// TIA Portal V19 export
DATA_BLOCK "DB_CommSlave"   // DB40
{ S7_Optimized_Access := 'TRUE' }
// stored: AutoNumber false, MemoryReserve 100
   VAR
      Left { ExternalAccessible := 'False'; ExternalVisible := 'False'; ExternalWritable := 'False'} : Struct
         xRobotHasStarted : Bool;   // Robot has started
         xRobotHasFinished : Bool;   // Robot has finished
         xBothSideFinished : Bool;   // Both robot finished
      END_STRUCT;
      Right { ExternalAccessible := 'False'; ExternalVisible := 'False'; ExternalWritable := 'False'} : Struct
         xRobotHasStarted : Bool;   // Robot has started
         xRobotHasFinished : Bool;   // Robot has finished
         xBothSideFinished : Bool;   // Both robot finished
      END_STRUCT;
   END_VAR
BEGIN
END_DATA_BLOCK
